# EPICS substitutions: evrSupport/Db/templates/archive_evr.substitutions
#
# EVR archive sample substitutions file
#
file archive_evr.template
{
	{	IOC	= $(IOC),	EVR	= $(EVR)	}
}
